# EPICS substitutions: db/Beckhoff_KL/ecmcBK1250.substitutions
file "ecmcEcSlave.template"
{
  pattern {}
          {}
}

file "ecmcBK1250.template"
{
  pattern {}
          {}
}
